TYPE ST_Feedback :
STRUCT
	em8000: ST_FeedbackStewart;
	em1500: ST_FeedbackStewart;
	mru1: ST_FeedbackMru;
	mru2: ST_FeedbackMru;
	comau: ST_FeedbackComau;
	winch: ST_FeedbackWinch;
	qtm: ST_FeedbackQualisys;
	at960: ST_FeedbackLeica;
END_STRUCT
END_TYPE

(* stored: Version 1.1.0.1, ProductVersion 3.1.4022.7
   DUT ST_Feedback: Id {c6e9113a-c1ff-4a71-b946-172d9bfe2bcf} *)
